GLOBALCONSTANTS DefaultPool_TC_SC_Numeric (* Numeric object pool constants (ID, Scale, Offset, Decimals) *)
  PACKAGE Uebungen::const::UT::TC_SC;
END_GLOBALCONSTANTS
